INTERFACE I_TriggerManager

METHOD GetAndResetTrigger
VAR_OUTPUT
    bLatchDetected : BOOL;
    nLatchTime_ns : ULINT; // [ns]
END_VAR
END_METHOD

END_INTERFACE

(* stored: Version 1.1.0.1
   Itf I_TriggerManager: Id {a096b8e4-37b6-42e8-9cff-ecc2fe66ae1d}
   Method GetAndResetTrigger: Id {3c1bd6da-2200-49ff-8c57-dca902b77851} *)
